FUNCTION F_NormVec4 : LREAL
VAR_INPUT
    iVec4 : I_Vec4;
END_VAR


F_NormVec4 := SQRT(F_NormSqVec4(iVec4));

END_FUNCTION

(* stored: Version 1.1.0.1
   POU F_NormVec4: Id {ac45f6af-5f3f-4ad4-9ea6-4799a1a4a160}, SpecialFunc None *)
